{attribute 'hide_all_locals'}
FUNCTION_BLOCK StopMoverGroup IMPLEMENTS ITask
VAR_INPUT
END_VAR
VAR_OUTPUT
END_VAR
VAR
	groupStop			: MC_GroupStop;
	_caGroup			: REFERENCE TO AXES_GROUP_REF;
	State: INT;
	_stopGroup : BOOL;
	_busy : BOOL;
	_error : BOOL;
	_done : BOOL;
	_jerk : MC_LREAL;
	_deceleration : MC_LREAL;
END_VAR

CASE State OF
	0:
		IF _stopGroup THEN
			_done := FALSE;
			_error := FALSE;
			_busy := TRUE;
			groupStop.Execute := TRUE;
			IF groupStop.Busy THEN
				State := 10;
				_stopGroup := FALSE;
			END_IF
		END_IF
	10:
		IF groupStop.Done THEN
			_done := TRUE;
		ELSIF groupStop.Error THEN
			_error := TRUE;
		END_IF
		IF _done OR _error THEN
			_busy := FALSE;
			groupStop.Execute := FALSE;
			State := 0;
		END_IF
END_CASE


groupStop(AxesGroup := _caGroup);

METHOD Abort : BOOL
groupStop.Execute := FALSE;
State := 0;
Abort := true;
END_METHOD

PROPERTY Busy : BOOL
GET
Busy := _busy;
END_GET
END_PROPERTY

PROPERTY PUBLIC Deceleration : MC_LREAL
GET
Deceleration := _deceleration;
END_GET
SET
_deceleration := Deceleration;
END_SET
END_PROPERTY

PROPERTY Done : BOOL
GET
Done := _done;
END_GET
END_PROPERTY

PROPERTY Error : BOOL
GET
Error := _error;
END_GET
END_PROPERTY

METHOD Execute : BOOL
_stopGroup := Execute := true;
END_METHOD

METHOD FB_init : BOOL
VAR_INPUT
	bInitRetains : BOOL; // if TRUE, the retain variables are initialized (warm start / cold start)
	bInCopyCode : BOOL;  // if TRUE, the instance afterwards gets moved into the copy code (online change)
	CAGroup : Reference TO AXES_GROUP_REF;
END_VAR
_caGroup REF= CAGroup;
END_METHOD

PROPERTY PUBLIC Jerk : MC_LREAL
GET
Jerk := _jerk;
END_GET
SET
_jerk := Jerk;
END_SET
END_PROPERTY

END_FUNCTION_BLOCK

(* stored: Version 1.1.0.1, ProductVersion 3.1.4024.6
   POU StopMoverGroup: Id {6b4de033-a9aa-4f32-b1bf-39cfc678fe0d}, SpecialFunc None
   Method Abort: Id {84d8ec1e-2daf-405f-97f6-3ca84d42d71e}
   Property Busy: Id {99d22da6-3624-4126-86aa-fd0d896ea214}
   Get Get: Id {c2285a56-2685-488d-b63e-c901e273fa49}
   Property Deceleration: Id {0004d781-7141-4b36-b997-4c91898ada85}
   Get Get: Id {7c555dbb-c240-433c-b2bd-142826283621}
   Set Set: Id {1d7070e8-d794-42ce-8f71-7d86bf122aa7}
   Property Done: Id {5fd3331a-3b67-41cd-869e-366d78814bd4}
   Get Get: Id {68dc2bb4-3cf0-4a53-9a59-1955c1d43eb0}
   Property Error: Id {6473f31d-8689-4f1d-b003-2cda08adf4bf}
   Get Get: Id {863dd496-99d1-42b2-80ad-3685c31ad1c2}
   Method Execute: Id {71f0bb1f-270a-4e16-bc2d-cde798c77078}
   Method FB_init: Id {4722d621-4f64-4e12-917c-563b1d0caeba}
   Property Jerk: Id {b1ff7d73-bcbe-4f76-8a44-8a6566f51dae}
   Get Get: Id {efa7d306-bb14-4089-980a-801ad7fc0442}
   Set Set: Id {f69d488a-866b-461e-9e2b-4eab77d736a0} *)
